// TIA Portal V18 export
// export: Created 2025-12-01T17:51:21.7919735Z, ExportSetting None, DisplayName Totally Integrated Automation Portal, DisplayVersion V18 Update 5, DisplayName TIA Portal Openness, DisplayVersion V18 Update 5, DisplayName TIA Portal Teamcenter Gateway, DisplayVersion V18, DisplayName TIA Portal Version Control Interface, DisplayVersion V18, DisplayName STEP 7 Professional, DisplayVersion V18 Update 5, DisplayName STEP 7 Safety, DisplayVersion V18, DisplayName WinCC Professional, DisplayVersion V18 Update 5
DATA_BLOCK "ST10_StopperCtrl_DB"   // DB2601
// stored: AutoNumber false, InstanceOfName ST10_StopperCtrl, InstanceOfType FB
"ST10_StopperCtrl"
   // VAR
   //    Stopper { S7_SetPoint := 'True'} : Array[1..100] of "StopperCtrl";
   // END_VAR
BEGIN
END_DATA_BLOCK
